TYPE EL5152_HWTOPLC :
	STRUCT
		
			channel1 : EL5152_HWTOPLC_PDOS;
			channel2 : EL5152_HWTOPLC_PDOS;

	END_STRUCT
END_TYPE

(* stored: Version 1.1.0.1
   DUT EL5152_HWTOPLC: Id {c5884e78-c61f-410f-9079-993a51b567a7} *)
